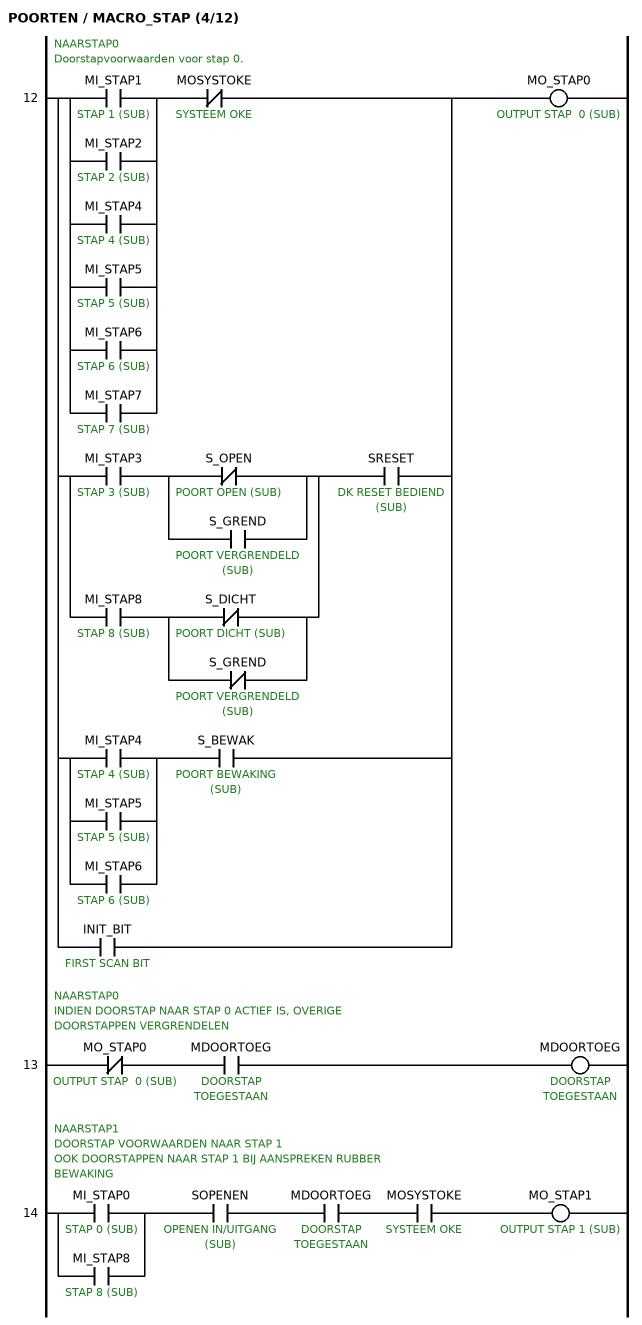
; [picture p469: POORTEN / MACRO_STAP, rungs 12-14]
; rung 12: NAARSTAP0 / Doorstapvoorwaarden voor stap 0.
LD MI_STAP1  ; STAP 1 (SUB)
OR MI_STAP2  ; STAP 2 (SUB)
OR MI_STAP4  ; STAP 4 (SUB)
OR MI_STAP5  ; STAP 5 (SUB)
OR MI_STAP6  ; STAP 6 (SUB)
OR MI_STAP7  ; STAP 7 (SUB)
ANDNOT MOSYSTOKE  ; SYSTEEM OKE
LD MI_STAP3  ; STAP 3 (SUB)
LDNOT S_OPEN  ; POORT OPEN (SUB)
OR S_GREND  ; POORT VERGRENDELD  (SUB)
ANDLD
LD MI_STAP8  ; STAP 8 (SUB)
LDNOT S_DICHT  ; POORT DICHT (SUB)
ORNOT S_GREND  ; POORT VERGRENDELD  (SUB)
ANDLD
ORLD
AND SRESET  ; DK RESET BEDIEND (SUB)
ORLD
LD MI_STAP4  ; STAP 4 (SUB)
OR MI_STAP5  ; STAP 5 (SUB)
OR MI_STAP6  ; STAP 6 (SUB)
AND S_BEWAK  ; POORT BEWAKING  (SUB)
ORLD
OR INIT_BIT  ; FIRST SCAN BIT
OUT MO_STAP0  ; OUTPUT STAP  0 (SUB)
; rung 13: NAARSTAP0 / INDIEN DOORSTAP NAAR STAP 0 ACTIEF IS, OVERIGE / DOORSTAPPEN VERGRENDELEN
LDNOT MO_STAP0  ; OUTPUT STAP  0 (SUB)
AND MDOORTOEG  ; DOORSTAP TOEGESTAAN
OUT MDOORTOEG  ; DOORSTAP TOEGESTAAN
; rung 14: NAARSTAP1 / DOORSTAP VOORWAARDEN NAAR STAP 1 / OOK DOORSTAPPEN NAAR STAP 1 BIJ AANSPREKEN RUBBER / BEWAKING
LD MI_STAP0  ; STAP 0 (SUB)
OR MI_STAP8  ; STAP 8 (SUB)
AND SOPENEN  ; OPENEN IN/UITGANG (SUB)
AND MDOORTOEG  ; DOORSTAP TOEGESTAAN
AND MOSYSTOKE  ; SYSTEEM OKE
OUT MO_STAP1  ; OUTPUT STAP 1 (SUB)

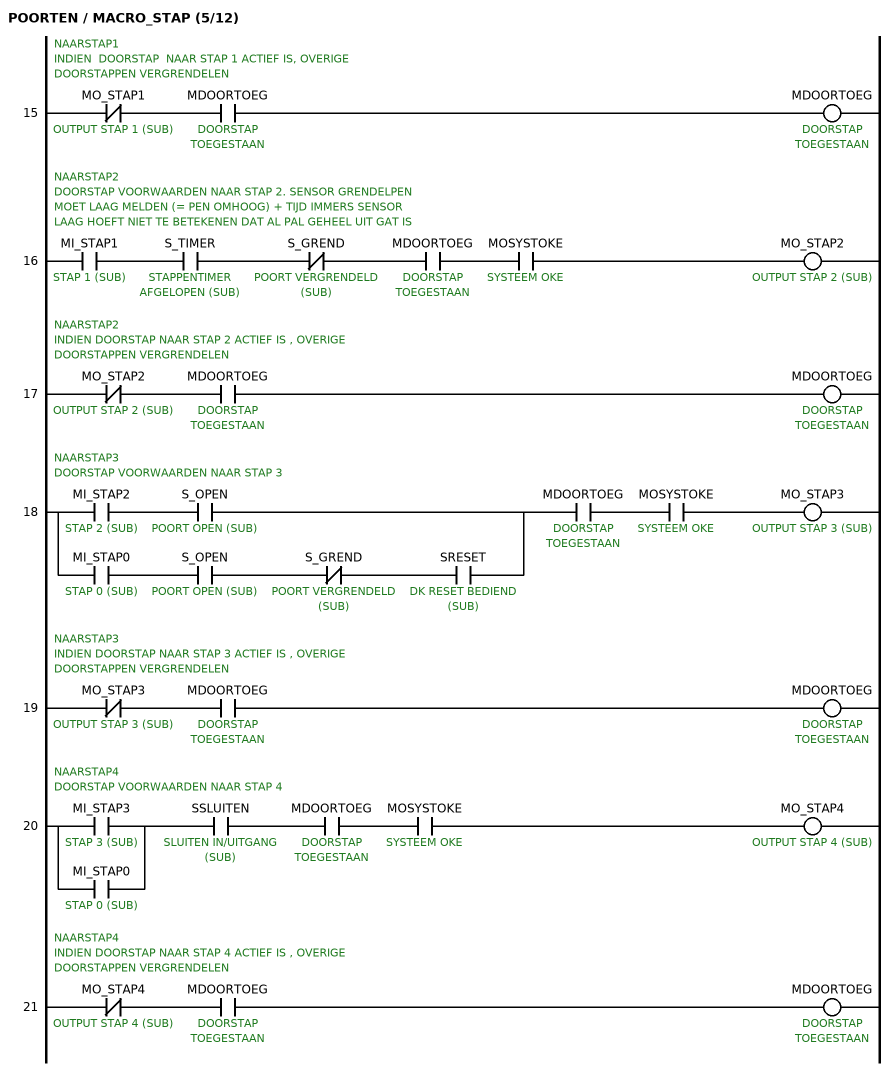
; rung 15: NAARSTAP1 / INDIEN  DOORSTAP  NAAR STAP 1 ACTIEF IS, OVERIGE / DOORSTAPPEN VERGRENDELEN
LDNOT MO_STAP1  ; OUTPUT STAP 1 (SUB)
AND MDOORTOEG  ; DOORSTAP TOEGESTAAN
OUT MDOORTOEG  ; DOORSTAP TOEGESTAAN
; rung 16: NAARSTAP2 / DOORSTAP VOORWAARDEN NAAR STAP 2. SENSOR GRENDELPEN / MOET LAAG MELDEN (= PEN OMHOOG) + TIJD IMMERS SENSOR / LAAG HOEFT NIET TE BETEKENEN DAT AL PAL GEHEEL UIT GAT IS
LD MI_STAP1  ; STAP 1 (SUB)
AND S_TIMER  ; STAPPENTIMER AFGELOPEN (SUB)
ANDNOT S_GREND  ; POORT VERGRENDELD  (SUB)
AND MDOORTOEG  ; DOORSTAP TOEGESTAAN
AND MOSYSTOKE  ; SYSTEEM OKE
OUT MO_STAP2  ; OUTPUT STAP 2 (SUB)
; rung 17: NAARSTAP2 / INDIEN DOORSTAP NAAR STAP 2 ACTIEF IS , OVERIGE / DOORSTAPPEN VERGRENDELEN
LDNOT MO_STAP2  ; OUTPUT STAP 2 (SUB)
AND MDOORTOEG  ; DOORSTAP TOEGESTAAN
OUT MDOORTOEG  ; DOORSTAP TOEGESTAAN
; rung 18: NAARSTAP3 / DOORSTAP VOORWAARDEN NAAR STAP 3
LD MI_STAP2  ; STAP 2 (SUB)
AND S_OPEN  ; POORT OPEN (SUB)
LD MI_STAP0  ; STAP 0 (SUB)
AND S_OPEN  ; POORT OPEN (SUB)
ANDNOT S_GREND  ; POORT VERGRENDELD  (SUB)
AND SRESET  ; DK RESET BEDIEND (SUB)
ORLD
AND MDOORTOEG  ; DOORSTAP TOEGESTAAN
AND MOSYSTOKE  ; SYSTEEM OKE
OUT MO_STAP3  ; OUTPUT STAP 3 (SUB)
; rung 19: NAARSTAP3 / INDIEN DOORSTAP NAAR STAP 3 ACTIEF IS , OVERIGE / DOORSTAPPEN VERGRENDELEN
LDNOT MO_STAP3  ; OUTPUT STAP 3 (SUB)
AND MDOORTOEG  ; DOORSTAP TOEGESTAAN
OUT MDOORTOEG  ; DOORSTAP TOEGESTAAN
; rung 20: NAARSTAP4 / DOORSTAP VOORWAARDEN NAAR STAP 4
LD MI_STAP3  ; STAP 3 (SUB)
OR MI_STAP0  ; STAP 0 (SUB)
AND SSLUITEN  ; SLUITEN IN/UITGANG (SUB)
AND MDOORTOEG  ; DOORSTAP TOEGESTAAN
AND MOSYSTOKE  ; SYSTEEM OKE
OUT MO_STAP4  ; OUTPUT STAP 4 (SUB)
; rung 21: NAARSTAP4 / INDIEN DOORSTAP NAAR STAP 4 ACTIEF IS , OVERIGE / DOORSTAPPEN VERGRENDELEN
LDNOT MO_STAP4  ; OUTPUT STAP 4 (SUB)
AND MDOORTOEG  ; DOORSTAP TOEGESTAAN
OUT MDOORTOEG  ; DOORSTAP TOEGESTAAN

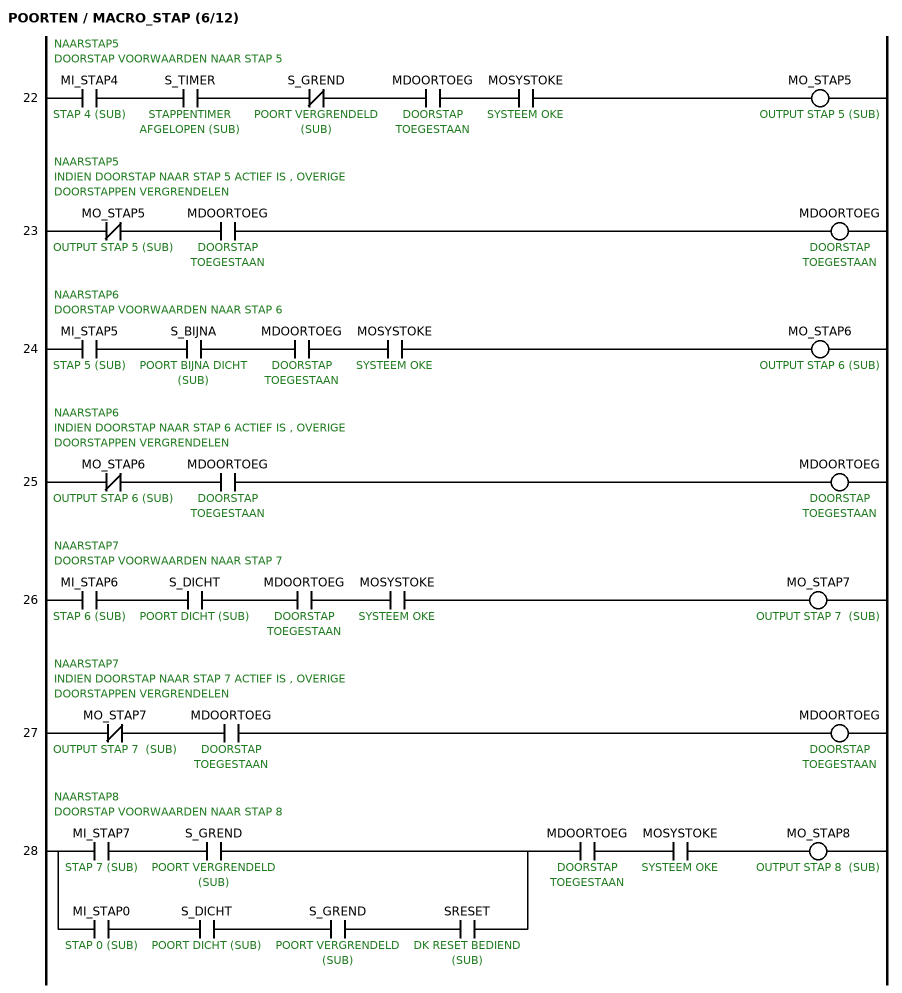
; rung 22: NAARSTAP5 / DOORSTAP VOORWAARDEN NAAR STAP 5
LD MI_STAP4  ; STAP 4 (SUB)
AND S_TIMER  ; STAPPENTIMER AFGELOPEN (SUB)
ANDNOT S_GREND  ; POORT VERGRENDELD  (SUB)
AND MDOORTOEG  ; DOORSTAP TOEGESTAAN
AND MOSYSTOKE  ; SYSTEEM OKE
OUT MO_STAP5  ; OUTPUT STAP 5 (SUB)
; rung 23: NAARSTAP5 / INDIEN DOORSTAP NAAR STAP 5 ACTIEF IS , OVERIGE / DOORSTAPPEN VERGRENDELEN
LDNOT MO_STAP5  ; OUTPUT STAP 5 (SUB)
AND MDOORTOEG  ; DOORSTAP TOEGESTAAN
OUT MDOORTOEG  ; DOORSTAP TOEGESTAAN
; rung 24: NAARSTAP6 / DOORSTAP VOORWAARDEN NAAR STAP 6
LD MI_STAP5  ; STAP 5 (SUB)
AND S_BIJNA  ; POORT BIJNA DICHT (SUB)
AND MDOORTOEG  ; DOORSTAP TOEGESTAAN
AND MOSYSTOKE  ; SYSTEEM OKE
OUT MO_STAP6  ; OUTPUT STAP 6 (SUB)
; rung 25: NAARSTAP6 / INDIEN DOORSTAP NAAR STAP 6 ACTIEF IS , OVERIGE / DOORSTAPPEN VERGRENDELEN
LDNOT MO_STAP6  ; OUTPUT STAP 6 (SUB)
AND MDOORTOEG  ; DOORSTAP TOEGESTAAN
OUT MDOORTOEG  ; DOORSTAP TOEGESTAAN
; rung 26: NAARSTAP7 / DOORSTAP VOORWAARDEN NAAR STAP 7
LD MI_STAP6  ; STAP 6 (SUB)
AND S_DICHT  ; POORT DICHT (SUB)
AND MDOORTOEG  ; DOORSTAP TOEGESTAAN
AND MOSYSTOKE  ; SYSTEEM OKE
OUT MO_STAP7  ; OUTPUT STAP 7  (SUB)
; rung 27: NAARSTAP7 / INDIEN DOORSTAP NAAR STAP 7 ACTIEF IS , OVERIGE / DOORSTAPPEN VERGRENDELEN
LDNOT MO_STAP7  ; OUTPUT STAP 7  (SUB)
AND MDOORTOEG  ; DOORSTAP TOEGESTAAN
OUT MDOORTOEG  ; DOORSTAP TOEGESTAAN
; rung 28: NAARSTAP8 / DOORSTAP VOORWAARDEN NAAR STAP 8
LD MI_STAP7  ; STAP 7 (SUB)
AND S_GREND  ; POORT VERGRENDELD  (SUB)
LD MI_STAP0  ; STAP 0 (SUB)
AND S_DICHT  ; POORT DICHT (SUB)
AND S_GREND  ; POORT VERGRENDELD  (SUB)
AND SRESET  ; DK RESET BEDIEND (SUB)
ORLD
AND MDOORTOEG  ; DOORSTAP TOEGESTAAN
AND MOSYSTOKE  ; SYSTEEM OKE
OUT MO_STAP8  ; OUTPUT STAP 8  (SUB)

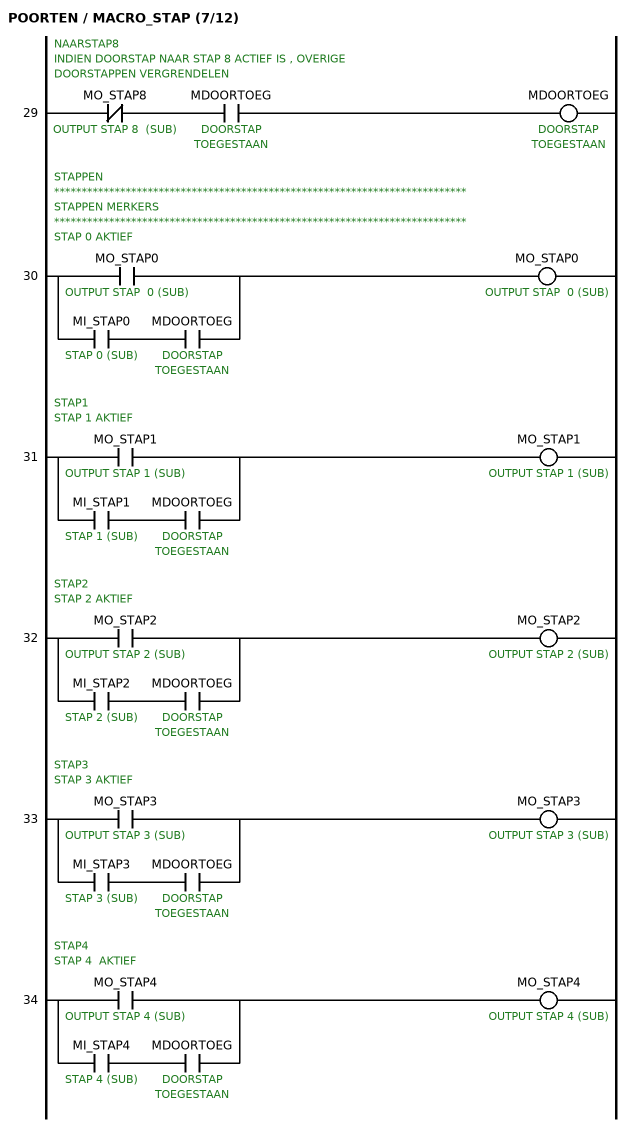
; rung 29: NAARSTAP8 / INDIEN DOORSTAP NAAR STAP 8 ACTIEF IS , OVERIGE / DOORSTAPPEN VERGRENDELEN
LDNOT MO_STAP8  ; OUTPUT STAP 8  (SUB)
AND MDOORTOEG  ; DOORSTAP TOEGESTAAN
OUT MDOORTOEG  ; DOORSTAP TOEGESTAAN
; rung 30: STAPPEN / *************************************************************************** / STAPPEN MERKERS / *************************************************************************** / STAP 0 AKTIEF
LD MO_STAP0  ; OUTPUT STAP  0 (SUB)
LD MI_STAP0  ; STAP 0 (SUB)
AND MDOORTOEG  ; DOORSTAP TOEGESTAAN
ORLD
OUT MO_STAP0  ; OUTPUT STAP  0 (SUB)
; rung 31: STAP1 / STAP 1 AKTIEF
LD MO_STAP1  ; OUTPUT STAP 1 (SUB)
LD MI_STAP1  ; STAP 1 (SUB)
AND MDOORTOEG  ; DOORSTAP TOEGESTAAN
ORLD
OUT MO_STAP1  ; OUTPUT STAP 1 (SUB)
; rung 32: STAP2 / STAP 2 AKTIEF
LD MO_STAP2  ; OUTPUT STAP 2 (SUB)
LD MI_STAP2  ; STAP 2 (SUB)
AND MDOORTOEG  ; DOORSTAP TOEGESTAAN
ORLD
OUT MO_STAP2  ; OUTPUT STAP 2 (SUB)
; rung 33: STAP3 / STAP 3 AKTIEF
LD MO_STAP3  ; OUTPUT STAP 3 (SUB)
LD MI_STAP3  ; STAP 3 (SUB)
AND MDOORTOEG  ; DOORSTAP TOEGESTAAN
ORLD
OUT MO_STAP3  ; OUTPUT STAP 3 (SUB)
; rung 34: STAP4 / STAP 4  AKTIEF
LD MO_STAP4  ; OUTPUT STAP 4 (SUB)
LD MI_STAP4  ; STAP 4 (SUB)
AND MDOORTOEG  ; DOORSTAP TOEGESTAAN
ORLD
OUT MO_STAP4  ; OUTPUT STAP 4 (SUB)

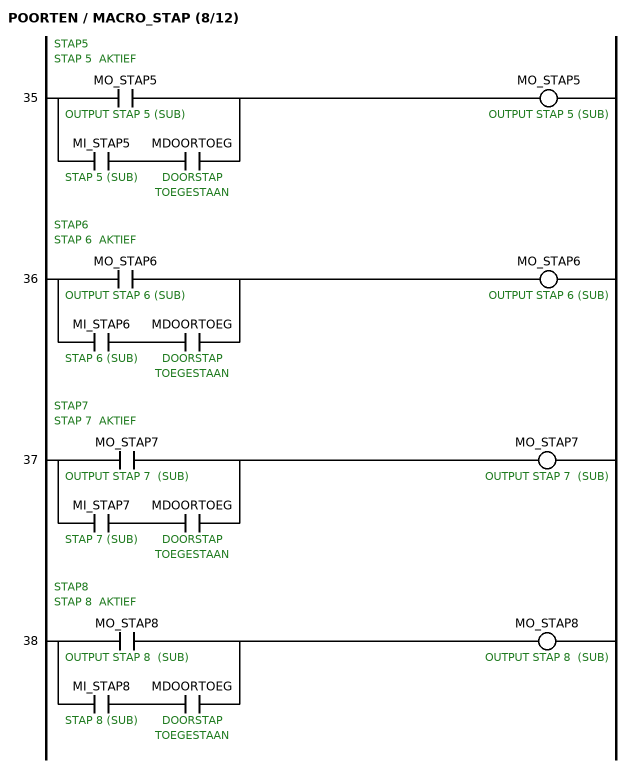
; rung 35: STAP5 / STAP 5  AKTIEF
LD MO_STAP5  ; OUTPUT STAP 5 (SUB)
LD MI_STAP5  ; STAP 5 (SUB)
AND MDOORTOEG  ; DOORSTAP TOEGESTAAN
ORLD
OUT MO_STAP5  ; OUTPUT STAP 5 (SUB)
; rung 36: STAP6 / STAP 6  AKTIEF
LD MO_STAP6  ; OUTPUT STAP 6 (SUB)
LD MI_STAP6  ; STAP 6 (SUB)
AND MDOORTOEG  ; DOORSTAP TOEGESTAAN
ORLD
OUT MO_STAP6  ; OUTPUT STAP 6 (SUB)
; rung 37: STAP7 / STAP 7  AKTIEF
LD MO_STAP7  ; OUTPUT STAP 7  (SUB)
LD MI_STAP7  ; STAP 7 (SUB)
AND MDOORTOEG  ; DOORSTAP TOEGESTAAN
ORLD
OUT MO_STAP7  ; OUTPUT STAP 7  (SUB)
; rung 38: STAP8 / STAP 8  AKTIEF
LD MO_STAP8  ; OUTPUT STAP 8  (SUB)
LD MI_STAP8  ; STAP 8 (SUB)
AND MDOORTOEG  ; DOORSTAP TOEGESTAAN
ORLD
OUT MO_STAP8  ; OUTPUT STAP 8  (SUB)

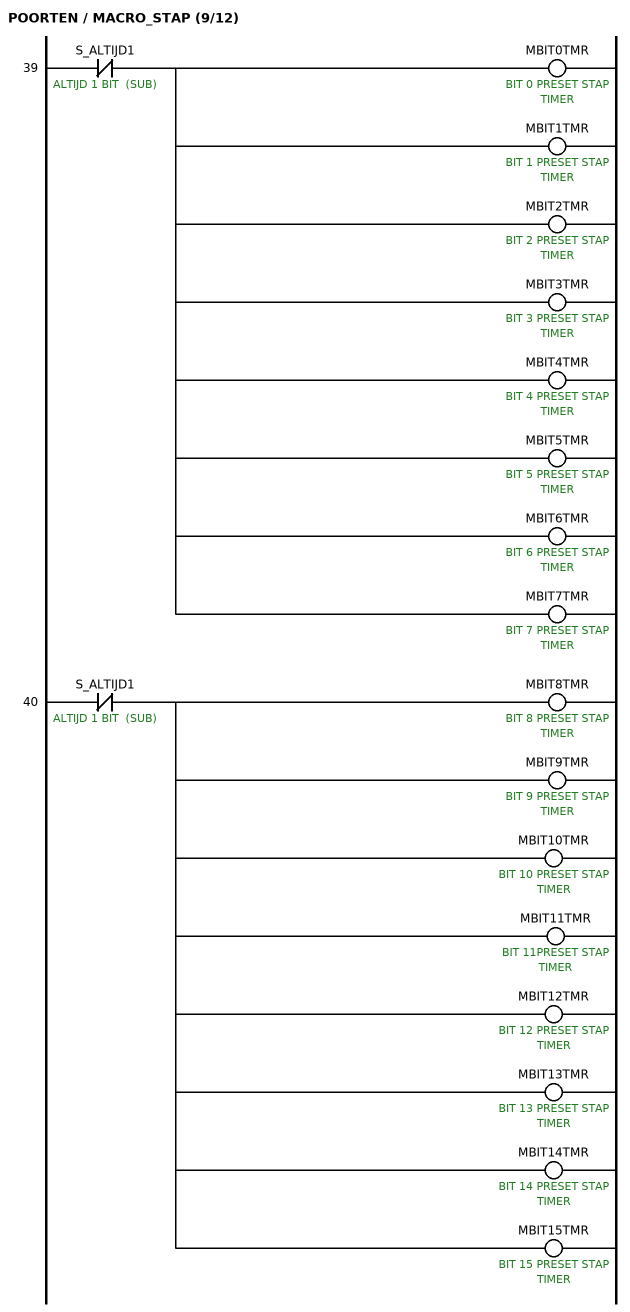
; rung 39
LDNOT S_ALTIJD1  ; ALTIJD 1 BIT  (SUB)
OUT MBIT0TMR  ; BIT 0 PRESET STAP TIMER
OUT MBIT1TMR  ; BIT 1 PRESET STAP TIMER
OUT MBIT2TMR  ; BIT 2 PRESET STAP TIMER
OUT MBIT3TMR  ; BIT 3 PRESET STAP TIMER
OUT MBIT4TMR  ; BIT 4 PRESET STAP TIMER
OUT MBIT5TMR  ; BIT 5 PRESET STAP TIMER
OUT MBIT6TMR  ; BIT 6 PRESET STAP TIMER
OUT MBIT7TMR  ; BIT 7 PRESET STAP TIMER
; rung 40
LDNOT S_ALTIJD1  ; ALTIJD 1 BIT  (SUB)
OUT MBIT8TMR  ; BIT 8 PRESET STAP TIMER
OUT MBIT9TMR  ; BIT 9 PRESET STAP TIMER
OUT MBIT10TMR  ; BIT 10 PRESET STAP TIMER
OUT MBIT11TMR  ; BIT 11PRESET STAP TIMER
OUT MBIT12TMR  ; BIT 12 PRESET STAP TIMER
OUT MBIT13TMR  ; BIT 13 PRESET STAP TIMER
OUT MBIT14TMR  ; BIT 14 PRESET STAP TIMER
OUT MBIT15TMR  ; BIT 15 PRESET STAP TIMER

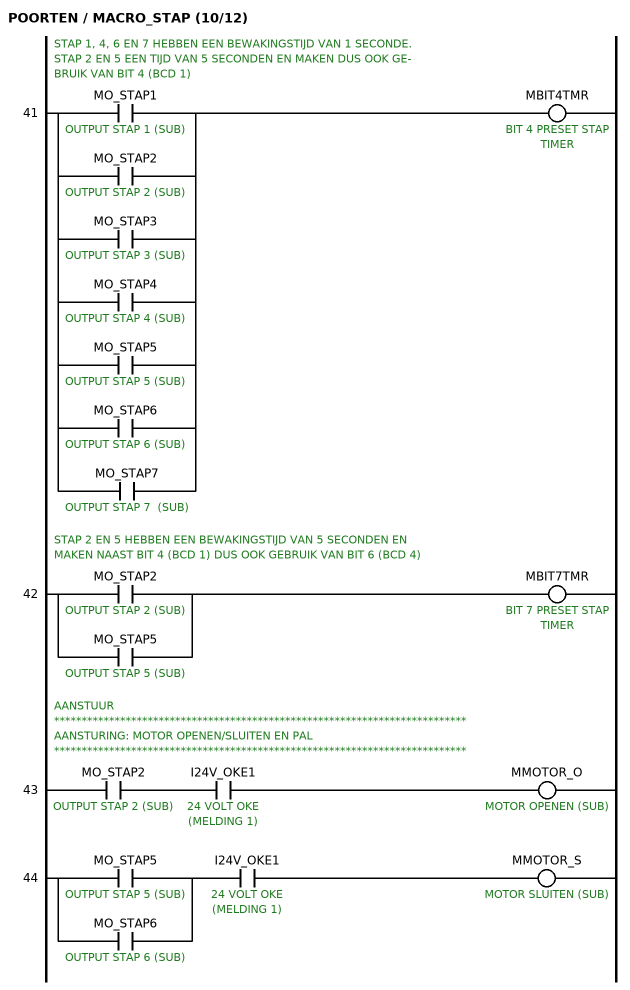
; rung 41: STAP 1, 4, 6 EN 7 HEBBEN EEN BEWAKINGSTIJD VAN 1 SECONDE. / STAP 2 EN 5 EEN TIJD VAN 5 SECONDEN EN MAKEN DUS OOK GE- / BRUIK VAN BIT 4 (BCD 1)
LD MO_STAP1  ; OUTPUT STAP 1 (SUB)
OR MO_STAP2  ; OUTPUT STAP 2 (SUB)
OR MO_STAP3  ; OUTPUT STAP 3 (SUB)
OR MO_STAP4  ; OUTPUT STAP 4 (SUB)
OR MO_STAP5  ; OUTPUT STAP 5 (SUB)
OR MO_STAP6  ; OUTPUT STAP 6 (SUB)
OR MO_STAP7  ; OUTPUT STAP 7  (SUB)
OUT MBIT4TMR  ; BIT 4 PRESET STAP TIMER
; rung 42: STAP 2 EN 5 HEBBEN EEN BEWAKINGSTIJD VAN 5 SECONDEN EN / MAKEN NAAST BIT 4 (BCD 1) DUS OOK GEBRUIK VAN BIT 6 (BCD 4)
LD MO_STAP2  ; OUTPUT STAP 2 (SUB)
OR MO_STAP5  ; OUTPUT STAP 5 (SUB)
OUT MBIT7TMR  ; BIT 7 PRESET STAP TIMER
; rung 43: AANSTUUR / *************************************************************************** / AANSTURING: MOTOR OPENEN/SLUITEN EN PAL / ***************************************************************************
LD MO_STAP2  ; OUTPUT STAP 2 (SUB)
AND I24V_OKE1  ; 24 VOLT OKE (MELDING 1)
OUT MMOTOR_O  ; MOTOR OPENEN (SUB)
; rung 44
LD MO_STAP5  ; OUTPUT STAP 5 (SUB)
OR MO_STAP6  ; OUTPUT STAP 6 (SUB)
AND I24V_OKE1  ; 24 VOLT OKE (MELDING 1)
OUT MMOTOR_S  ; MOTOR SLUITEN (SUB)

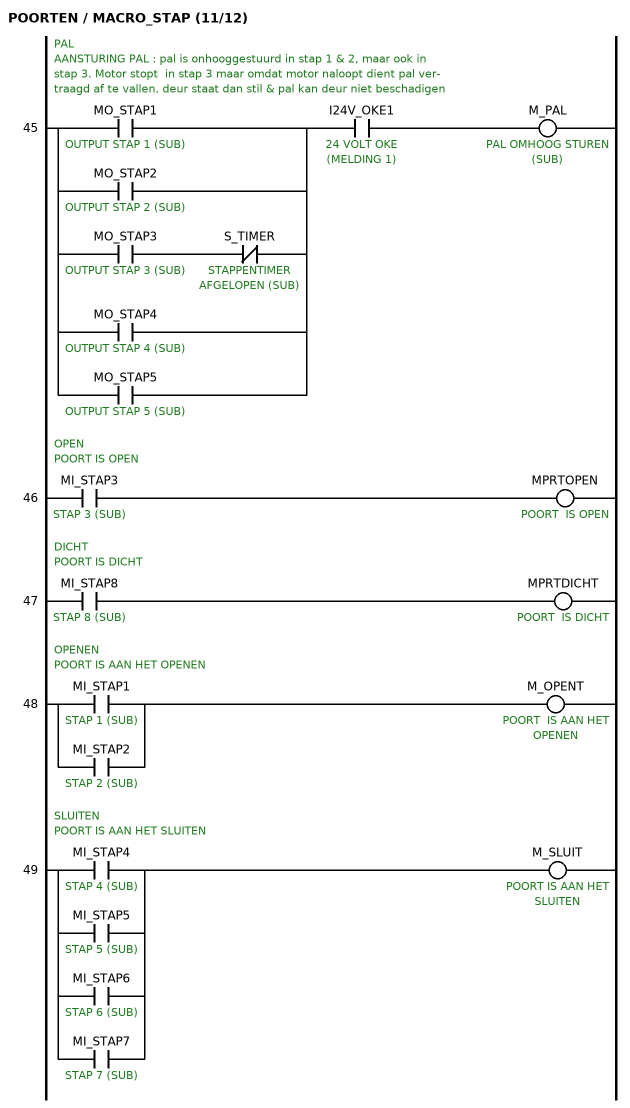
; rung 45: PAL / AANSTURING PAL : pal is onhooggestuurd in stap 1 & 2, maar ook in / stap 3. Motor stopt  in stap 3 maar omdat motor naloopt dient pal ver- / traagd af te vallen. deur staat dan stil & pal kan deur niet beschadigen
LD MO_STAP1  ; OUTPUT STAP 1 (SUB)
OR MO_STAP2  ; OUTPUT STAP 2 (SUB)
LD MO_STAP3  ; OUTPUT STAP 3 (SUB)
ANDNOT S_TIMER  ; STAPPENTIMER AFGELOPEN (SUB)
ORLD
OR MO_STAP4  ; OUTPUT STAP 4 (SUB)
OR MO_STAP5  ; OUTPUT STAP 5 (SUB)
AND I24V_OKE1  ; 24 VOLT OKE (MELDING 1)
OUT M_PAL  ; PAL OMHOOG STUREN (SUB)
; rung 46: OPEN / POORT IS OPEN
LD MI_STAP3  ; STAP 3 (SUB)
OUT MPRTOPEN  ; POORT  IS OPEN
; rung 47: DICHT / POORT IS DICHT
LD MI_STAP8  ; STAP 8 (SUB)
OUT MPRTDICHT  ; POORT  IS DICHT
; rung 48: OPENEN / POORT IS AAN HET OPENEN
LD MI_STAP1  ; STAP 1 (SUB)
OR MI_STAP2  ; STAP 2 (SUB)
OUT M_OPENT  ; POORT  IS AAN HET OPENEN
; rung 49: SLUITEN / POORT IS AAN HET SLUITEN
LD MI_STAP4  ; STAP 4 (SUB)
OR MI_STAP5  ; STAP 5 (SUB)
OR MI_STAP6  ; STAP 6 (SUB)
OR MI_STAP7  ; STAP 7 (SUB)
OUT M_SLUIT  ; POORT IS AAN HET SLUITEN

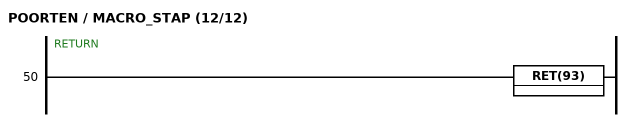
; rung 50: RETURN
RET(93)

### Section SUB_DISPLAY

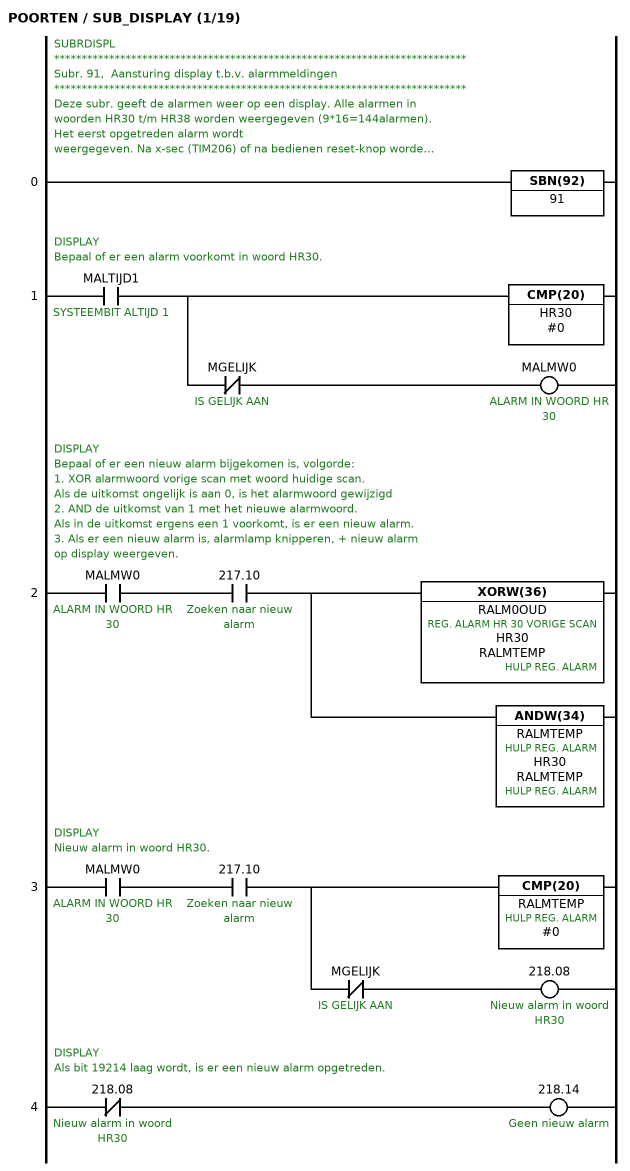
; rung 0: SUBRDISPL / *************************************************************************** / Subr. 91,  Aansturing display t.b.v. alarmmeldingen / *************************************************************************** / Deze subr. geeft de alarmen weer op een display. Alle alarmen in / woorden HR30 t/m HR38 worden weergegeven (9*16=144alarmen). / Het eerst opgetreden alarm wordt / weergegeven. Na x-sec (TIM206) of na bedienen reset-knop worden / alle alarmen gescrolld, met schroltijd TIM207. Als tijdens scrollen een / nieuw alarm optreedt, wordt dit alarm weer continu weergegeven.
SBN(92) 91
; rung 1: DISPLAY / Bepaal of er een alarm voorkomt in woord HR30.
LD MALTIJD1  ; SYSTEEMBIT ALTIJD 1
CMP(20) HR30 #0
ANDNOT MGELIJK  ; IS GELIJK AAN
OUT MALMW0  ; ALARM IN WOORD HR 30
; rung 2: DISPLAY / Bepaal of er een nieuw alarm bijgekomen is, volgorde: / 1. XOR alarmwoord vorige scan met woord huidige scan. / Als de uitkomst ongelijk is aan 0, is het alarmwoord gewijzigd / 2. AND de uitkomst van 1 met het nieuwe alarmwoord. / Als in de uitkomst ergens een 1 voorkomt, is er een nieuw alarm. / 3. Als er een nieuw alarm is, alarmlamp knipperen, + nieuw alarm / op display weergeven.
LD MALMW0  ; ALARM IN WOORD HR 30
AND 217.10  ; Zoeken naar nieuw alarm
XORW(36) RALM0OUD HR30 RALMTEMP  ; REG. ALARM HR 30 VORIGE SCAN, HULP REG. ALARM
ANDW(34) RALMTEMP HR30 RALMTEMP  ; HULP REG. ALARM
; rung 3: DISPLAY / Nieuw alarm in woord HR30.
LD MALMW0  ; ALARM IN WOORD HR 30
AND 217.10  ; Zoeken naar nieuw alarm
CMP(20) RALMTEMP #0  ; HULP REG. ALARM
ANDNOT MGELIJK  ; IS GELIJK AAN
OUT 218.08  ; Nieuw alarm in woord HR30
; rung 4: DISPLAY / Als bit 19214 laag wordt, is er een nieuw alarm opgetreden.
LDNOT 218.08  ; Nieuw alarm in woord HR30
OUT 218.14  ; Geen nieuw alarm

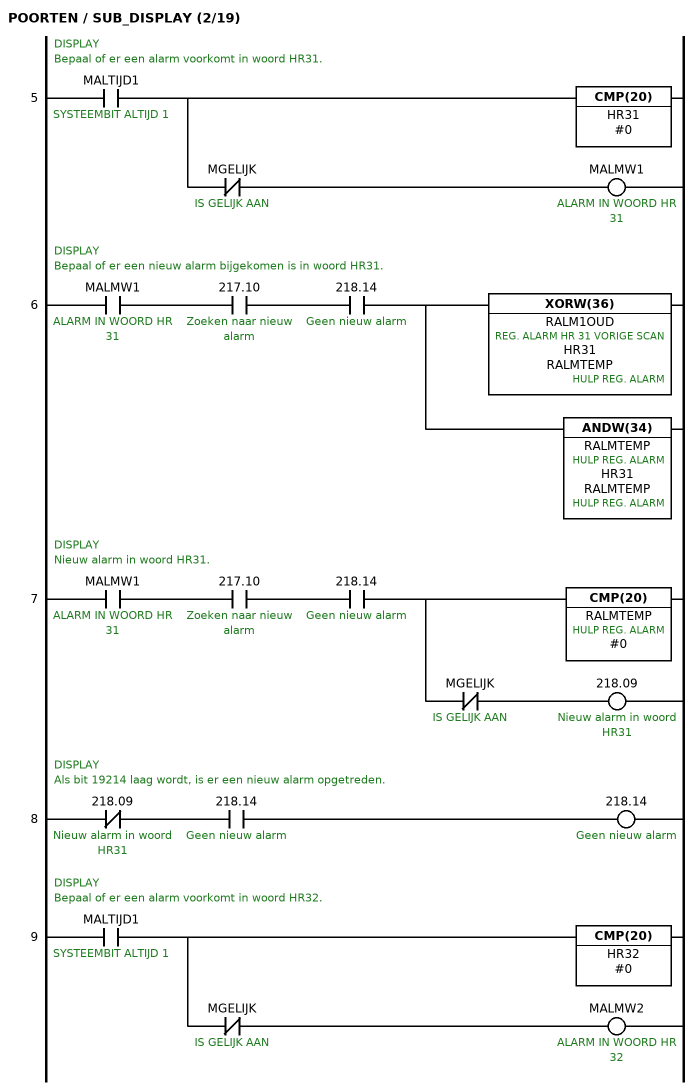
; rung 5: DISPLAY / Bepaal of er een alarm voorkomt in woord HR31.
LD MALTIJD1  ; SYSTEEMBIT ALTIJD 1
CMP(20) HR31 #0
ANDNOT MGELIJK  ; IS GELIJK AAN
OUT MALMW1  ; ALARM IN WOORD HR 31
; rung 6: DISPLAY / Bepaal of er een nieuw alarm bijgekomen is in woord HR31.
LD MALMW1  ; ALARM IN WOORD HR 31
AND 217.10  ; Zoeken naar nieuw alarm
AND 218.14  ; Geen nieuw alarm
XORW(36) RALM1OUD HR31 RALMTEMP  ; REG. ALARM HR 31 VORIGE SCAN, HULP REG. ALARM
ANDW(34) RALMTEMP HR31 RALMTEMP  ; HULP REG. ALARM
; rung 7: DISPLAY / Nieuw alarm in woord HR31.
LD MALMW1  ; ALARM IN WOORD HR 31
AND 217.10  ; Zoeken naar nieuw alarm
AND 218.14  ; Geen nieuw alarm
CMP(20) RALMTEMP #0  ; HULP REG. ALARM
ANDNOT MGELIJK  ; IS GELIJK AAN
OUT 218.09  ; Nieuw alarm in woord HR31
; rung 8: DISPLAY / Als bit 19214 laag wordt, is er een nieuw alarm opgetreden.
LDNOT 218.09  ; Nieuw alarm in woord HR31
AND 218.14  ; Geen nieuw alarm
OUT 218.14  ; Geen nieuw alarm
; rung 9: DISPLAY / Bepaal of er een alarm voorkomt in woord HR32.
LD MALTIJD1  ; SYSTEEMBIT ALTIJD 1
CMP(20) HR32 #0
ANDNOT MGELIJK  ; IS GELIJK AAN
OUT MALMW2  ; ALARM IN WOORD HR 32

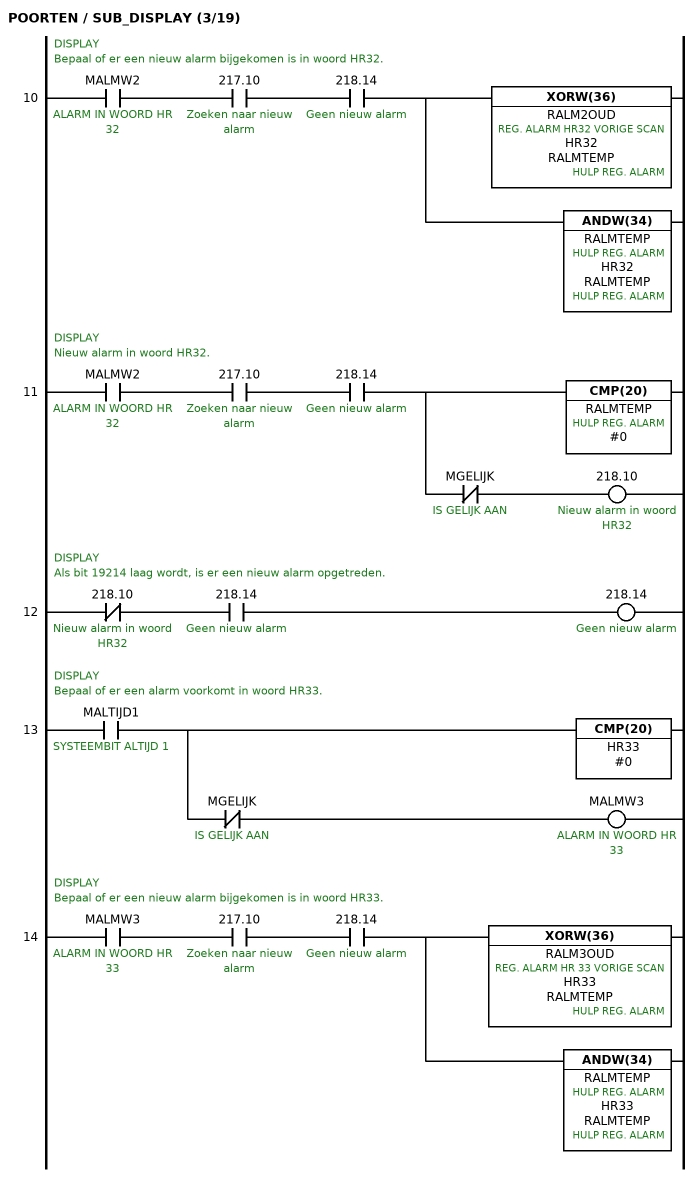
; rung 10: DISPLAY / Bepaal of er een nieuw alarm bijgekomen is in woord HR32.
LD MALMW2  ; ALARM IN WOORD HR 32
AND 217.10  ; Zoeken naar nieuw alarm
AND 218.14  ; Geen nieuw alarm
XORW(36) RALM2OUD HR32 RALMTEMP  ; REG. ALARM HR32 VORIGE SCAN, HULP REG. ALARM
ANDW(34) RALMTEMP HR32 RALMTEMP  ; HULP REG. ALARM
; rung 11: DISPLAY / Nieuw alarm in woord HR32.
LD MALMW2  ; ALARM IN WOORD HR 32
AND 217.10  ; Zoeken naar nieuw alarm
AND 218.14  ; Geen nieuw alarm
CMP(20) RALMTEMP #0  ; HULP REG. ALARM
ANDNOT MGELIJK  ; IS GELIJK AAN
OUT 218.10  ; Nieuw alarm in woord HR32
; rung 12: DISPLAY / Als bit 19214 laag wordt, is er een nieuw alarm opgetreden.
LDNOT 218.10  ; Nieuw alarm in woord HR32
AND 218.14  ; Geen nieuw alarm
OUT 218.14  ; Geen nieuw alarm
; rung 13: DISPLAY / Bepaal of er een alarm voorkomt in woord HR33.
LD MALTIJD1  ; SYSTEEMBIT ALTIJD 1
CMP(20) HR33 #0
ANDNOT MGELIJK  ; IS GELIJK AAN
OUT MALMW3  ; ALARM IN WOORD HR 33
; rung 14: DISPLAY / Bepaal of er een nieuw alarm bijgekomen is in woord HR33.
LD MALMW3  ; ALARM IN WOORD HR 33
AND 217.10  ; Zoeken naar nieuw alarm
AND 218.14  ; Geen nieuw alarm
XORW(36) RALM3OUD HR33 RALMTEMP  ; REG. ALARM HR 33 VORIGE SCAN, HULP REG. ALARM
ANDW(34) RALMTEMP HR33 RALMTEMP  ; HULP REG. ALARM

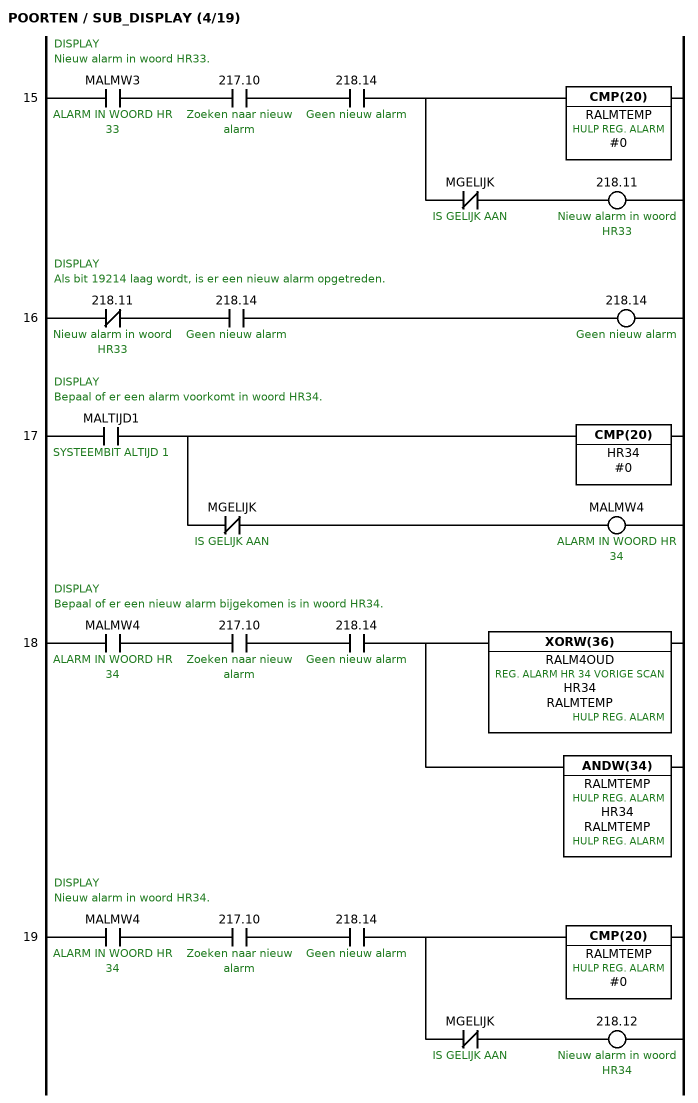
; rung 15: DISPLAY / Nieuw alarm in woord HR33.
LD MALMW3  ; ALARM IN WOORD HR 33
AND 217.10  ; Zoeken naar nieuw alarm
AND 218.14  ; Geen nieuw alarm
CMP(20) RALMTEMP #0  ; HULP REG. ALARM
ANDNOT MGELIJK  ; IS GELIJK AAN
OUT 218.11  ; Nieuw alarm in woord HR33
; rung 16: DISPLAY / Als bit 19214 laag wordt, is er een nieuw alarm opgetreden.
LDNOT 218.11  ; Nieuw alarm in woord HR33
AND 218.14  ; Geen nieuw alarm
OUT 218.14  ; Geen nieuw alarm
; rung 17: DISPLAY / Bepaal of er een alarm voorkomt in woord HR34.
LD MALTIJD1  ; SYSTEEMBIT ALTIJD 1
CMP(20) HR34 #0
ANDNOT MGELIJK  ; IS GELIJK AAN
OUT MALMW4  ; ALARM IN WOORD HR 34
; rung 18: DISPLAY / Bepaal of er een nieuw alarm bijgekomen is in woord HR34.
LD MALMW4  ; ALARM IN WOORD HR 34
AND 217.10  ; Zoeken naar nieuw alarm
AND 218.14  ; Geen nieuw alarm
XORW(36) RALM4OUD HR34 RALMTEMP  ; REG. ALARM HR 34 VORIGE SCAN, HULP REG. ALARM
ANDW(34) RALMTEMP HR34 RALMTEMP  ; HULP REG. ALARM
; rung 19: DISPLAY / Nieuw alarm in woord HR34.
LD MALMW4  ; ALARM IN WOORD HR 34
AND 217.10  ; Zoeken naar nieuw alarm
AND 218.14  ; Geen nieuw alarm
CMP(20) RALMTEMP #0  ; HULP REG. ALARM
ANDNOT MGELIJK  ; IS GELIJK AAN
OUT 218.12  ; Nieuw alarm in woord HR34

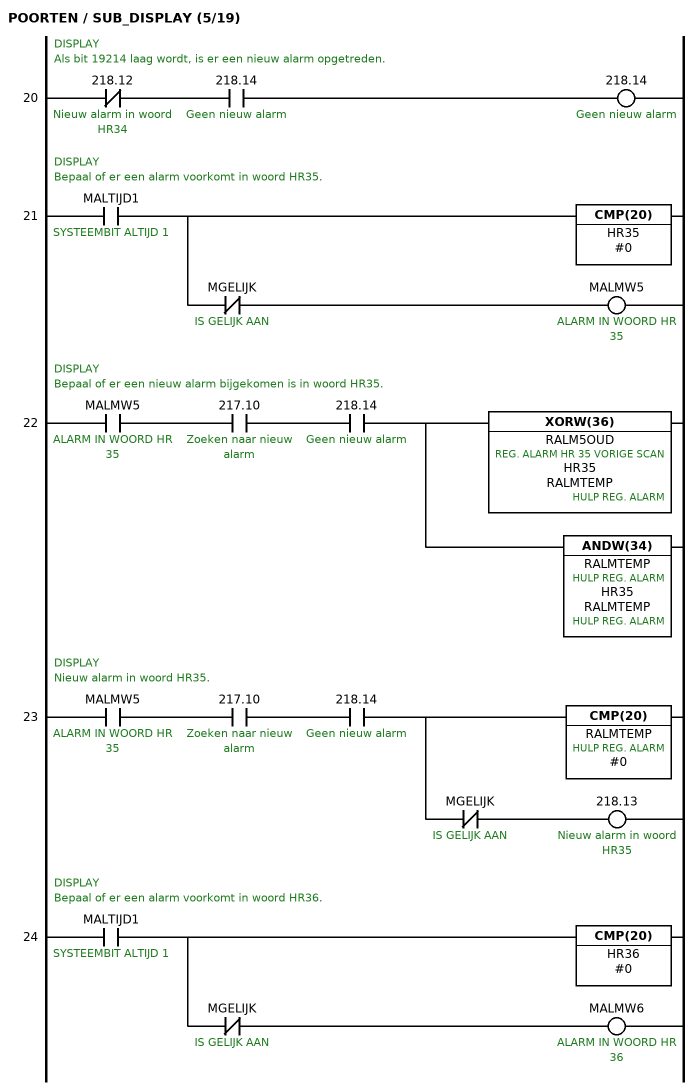
; rung 20: DISPLAY / Als bit 19214 laag wordt, is er een nieuw alarm opgetreden.
LDNOT 218.12  ; Nieuw alarm in woord HR34
AND 218.14  ; Geen nieuw alarm
OUT 218.14  ; Geen nieuw alarm
; rung 21: DISPLAY / Bepaal of er een alarm voorkomt in woord HR35.
LD MALTIJD1  ; SYSTEEMBIT ALTIJD 1
CMP(20) HR35 #0
ANDNOT MGELIJK  ; IS GELIJK AAN
OUT MALMW5  ; ALARM IN WOORD HR 35
; rung 22: DISPLAY / Bepaal of er een nieuw alarm bijgekomen is in woord HR35.
LD MALMW5  ; ALARM IN WOORD HR 35
AND 217.10  ; Zoeken naar nieuw alarm
AND 218.14  ; Geen nieuw alarm
XORW(36) RALM5OUD HR35 RALMTEMP  ; REG. ALARM HR 35 VORIGE SCAN, HULP REG. ALARM
ANDW(34) RALMTEMP HR35 RALMTEMP  ; HULP REG. ALARM
; rung 23: DISPLAY / Nieuw alarm in woord HR35.
LD MALMW5  ; ALARM IN WOORD HR 35
AND 217.10  ; Zoeken naar nieuw alarm
AND 218.14  ; Geen nieuw alarm
CMP(20) RALMTEMP #0  ; HULP REG. ALARM
ANDNOT MGELIJK  ; IS GELIJK AAN
OUT 218.13  ; Nieuw alarm in woord HR35
; rung 24: DISPLAY / Bepaal of er een alarm voorkomt in woord HR36.
LD MALTIJD1  ; SYSTEEMBIT ALTIJD 1
CMP(20) HR36 #0
ANDNOT MGELIJK  ; IS GELIJK AAN
OUT MALMW6  ; ALARM IN WOORD HR 36

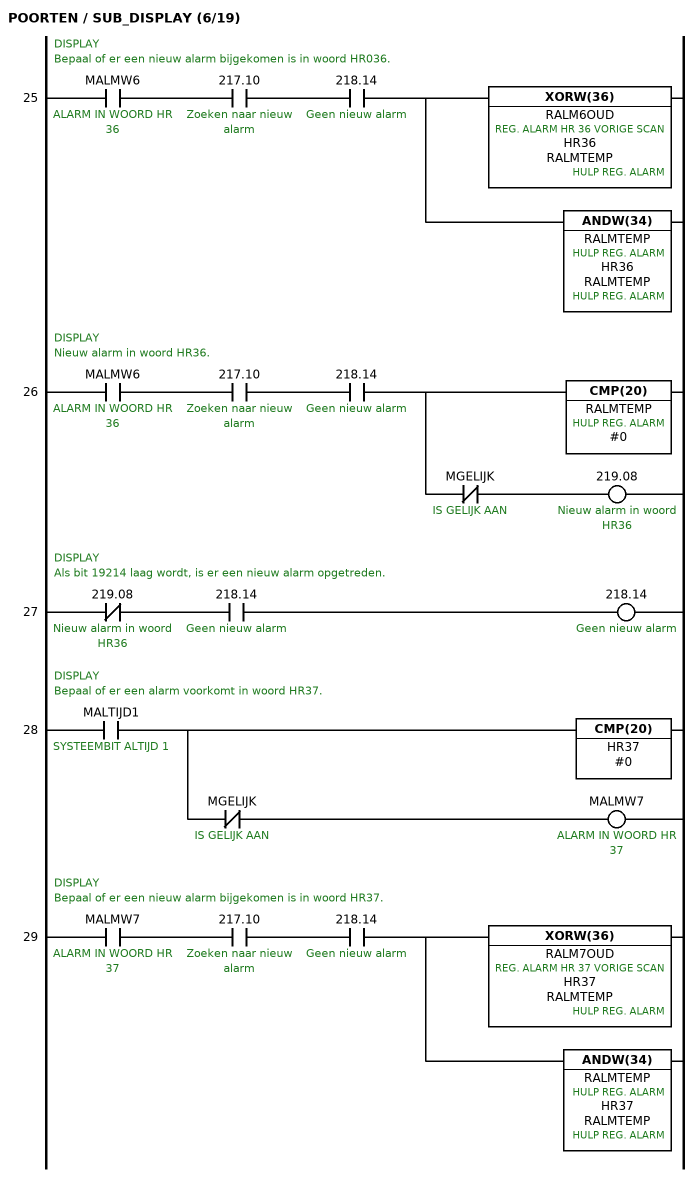
; rung 25: DISPLAY / Bepaal of er een nieuw alarm bijgekomen is in woord HR036.
LD MALMW6  ; ALARM IN WOORD HR 36
AND 217.10  ; Zoeken naar nieuw alarm
AND 218.14  ; Geen nieuw alarm
XORW(36) RALM6OUD HR36 RALMTEMP  ; REG. ALARM HR 36 VORIGE SCAN, HULP REG. ALARM
ANDW(34) RALMTEMP HR36 RALMTEMP  ; HULP REG. ALARM
; rung 26: DISPLAY / Nieuw alarm in woord HR36.
LD MALMW6  ; ALARM IN WOORD HR 36
AND 217.10  ; Zoeken naar nieuw alarm
AND 218.14  ; Geen nieuw alarm
CMP(20) RALMTEMP #0  ; HULP REG. ALARM
ANDNOT MGELIJK  ; IS GELIJK AAN
OUT 219.08  ; Nieuw alarm in woord HR36
; rung 27: DISPLAY / Als bit 19214 laag wordt, is er een nieuw alarm opgetreden.
LDNOT 219.08  ; Nieuw alarm in woord HR36
AND 218.14  ; Geen nieuw alarm
OUT 218.14  ; Geen nieuw alarm
; rung 28: DISPLAY / Bepaal of er een alarm voorkomt in woord HR37.
LD MALTIJD1  ; SYSTEEMBIT ALTIJD 1
CMP(20) HR37 #0
ANDNOT MGELIJK  ; IS GELIJK AAN
OUT MALMW7  ; ALARM IN WOORD HR 37
; rung 29: DISPLAY / Bepaal of er een nieuw alarm bijgekomen is in woord HR37.
LD MALMW7  ; ALARM IN WOORD HR 37
AND 217.10  ; Zoeken naar nieuw alarm
AND 218.14  ; Geen nieuw alarm
XORW(36) RALM7OUD HR37 RALMTEMP  ; REG. ALARM HR 37 VORIGE SCAN, HULP REG. ALARM
ANDW(34) RALMTEMP HR37 RALMTEMP  ; HULP REG. ALARM

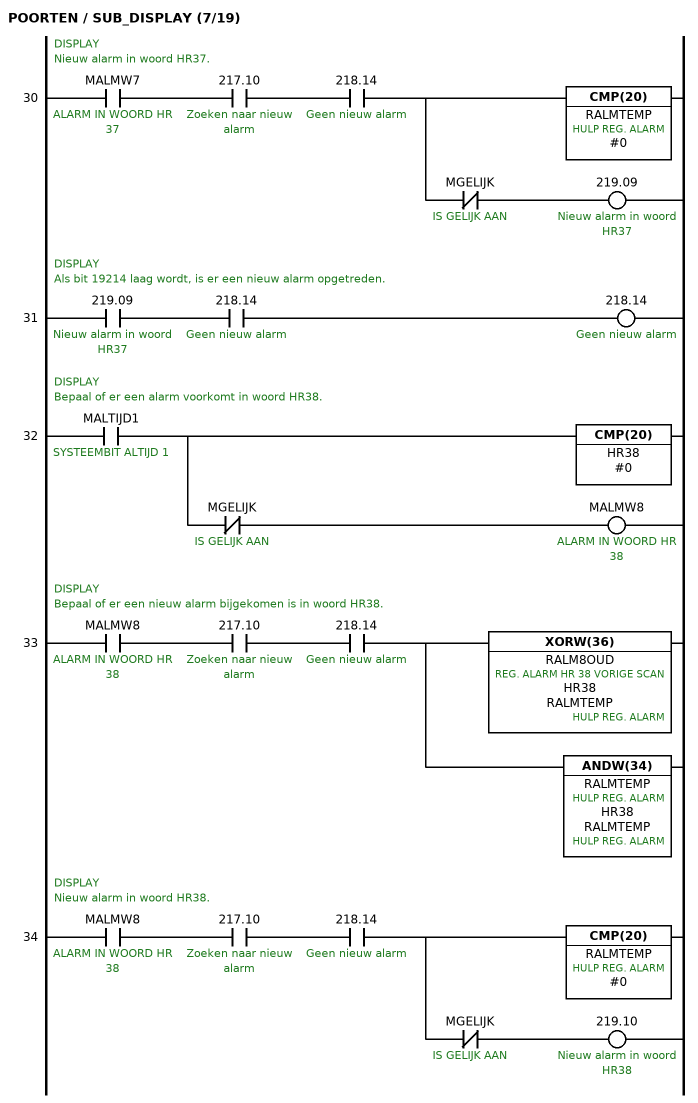
; rung 30: DISPLAY / Nieuw alarm in woord HR37.
LD MALMW7  ; ALARM IN WOORD HR 37
AND 217.10  ; Zoeken naar nieuw alarm
AND 218.14  ; Geen nieuw alarm
CMP(20) RALMTEMP #0  ; HULP REG. ALARM
ANDNOT MGELIJK  ; IS GELIJK AAN
OUT 219.09  ; Nieuw alarm in woord HR37
; rung 31: DISPLAY / Als bit 19214 laag wordt, is er een nieuw alarm opgetreden.
LD 219.09  ; Nieuw alarm in woord HR37
AND 218.14  ; Geen nieuw alarm
OUT 218.14  ; Geen nieuw alarm
; rung 32: DISPLAY / Bepaal of er een alarm voorkomt in woord HR38.
LD MALTIJD1  ; SYSTEEMBIT ALTIJD 1
CMP(20) HR38 #0
ANDNOT MGELIJK  ; IS GELIJK AAN
OUT MALMW8  ; ALARM IN WOORD HR 38
; rung 33: DISPLAY / Bepaal of er een nieuw alarm bijgekomen is in woord HR38.
LD MALMW8  ; ALARM IN WOORD HR 38
AND 217.10  ; Zoeken naar nieuw alarm
AND 218.14  ; Geen nieuw alarm
XORW(36) RALM8OUD HR38 RALMTEMP  ; REG. ALARM HR 38 VORIGE SCAN, HULP REG. ALARM
ANDW(34) RALMTEMP HR38 RALMTEMP  ; HULP REG. ALARM
; rung 34: DISPLAY / Nieuw alarm in woord HR38.
LD MALMW8  ; ALARM IN WOORD HR 38
AND 217.10  ; Zoeken naar nieuw alarm
AND 218.14  ; Geen nieuw alarm
CMP(20) RALMTEMP #0  ; HULP REG. ALARM
ANDNOT MGELIJK  ; IS GELIJK AAN
OUT 219.10  ; Nieuw alarm in woord HR38

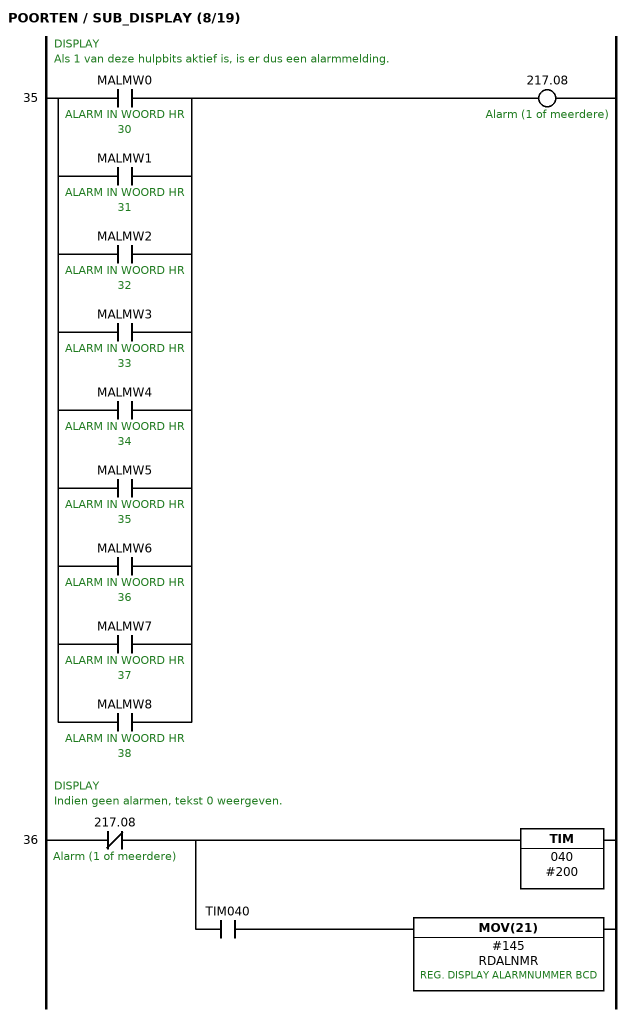
; rung 35: DISPLAY / Als 1 van deze hulpbits aktief is, is er dus een alarmmelding.
LD MALMW0  ; ALARM IN WOORD HR 30
OR MALMW1  ; ALARM IN WOORD HR 31
OR MALMW2  ; ALARM IN WOORD HR 32
OR MALMW3  ; ALARM IN WOORD HR 33
OR MALMW4  ; ALARM IN WOORD HR 34
OR MALMW5  ; ALARM IN WOORD HR 35
OR MALMW6  ; ALARM IN WOORD HR 36
OR MALMW7  ; ALARM IN WOORD HR 37
OR MALMW8  ; ALARM IN WOORD HR 38
OUT 217.08  ; Alarm (1 of meerdere)
; rung 36: DISPLAY / Indien geen alarmen, tekst 0 weergeven.
LDNOT 217.08  ; Alarm (1 of meerdere)
TIM 040 #200
AND TIM040
MOV(21) #145 RDALNMR  ; REG. DISPLAY ALARMNUMMER BCD

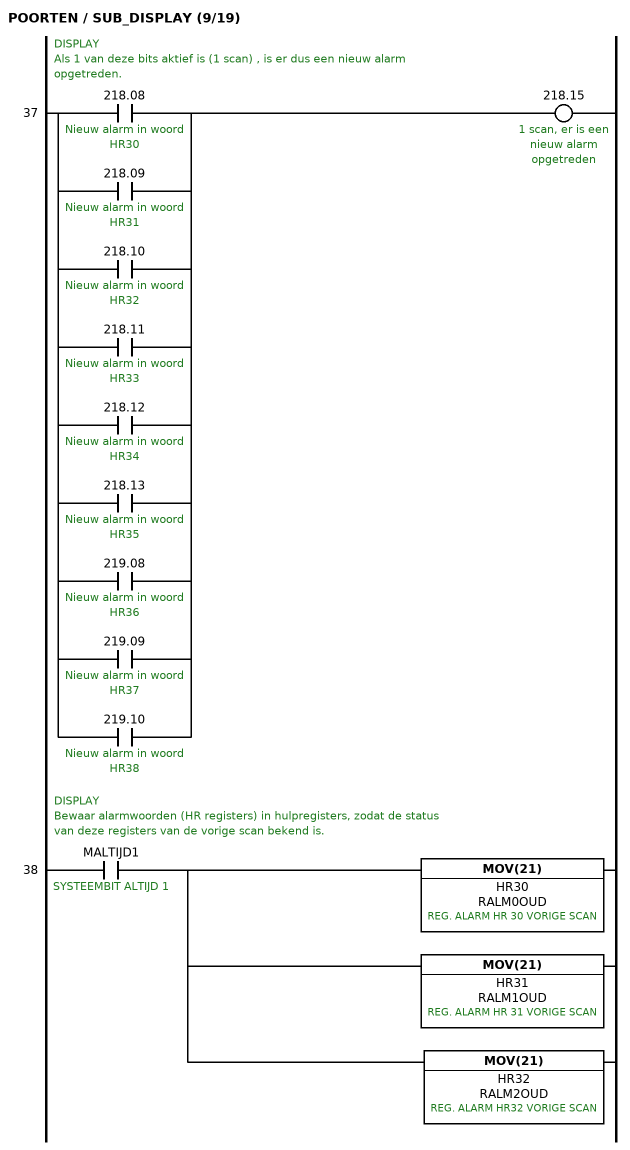
; rung 37: DISPLAY / Als 1 van deze bits aktief is (1 scan) , is er dus een nieuw alarm / opgetreden.
LD 218.08  ; Nieuw alarm in woord HR30
OR 218.09  ; Nieuw alarm in woord HR31
OR 218.10  ; Nieuw alarm in woord HR32
OR 218.11  ; Nieuw alarm in woord HR33
OR 218.12  ; Nieuw alarm in woord HR34
OR 218.13  ; Nieuw alarm in woord HR35
OR 219.08  ; Nieuw alarm in woord HR36
OR 219.09  ; Nieuw alarm in woord HR37
OR 219.10  ; Nieuw alarm in woord HR38
OUT 218.15  ; 1 scan, er is een nieuw alarm opgetreden
; rung 38: DISPLAY / Bewaar alarmwoorden (HR registers) in hulpregisters, zodat de status / van deze registers van de vorige scan bekend is.
LD MALTIJD1  ; SYSTEEMBIT ALTIJD 1
MOV(21) HR30 RALM0OUD  ; REG. ALARM HR 30 VORIGE SCAN
MOV(21) HR31 RALM1OUD  ; REG. ALARM HR 31 VORIGE SCAN
MOV(21) HR32 RALM2OUD  ; REG. ALARM HR32 VORIGE SCAN

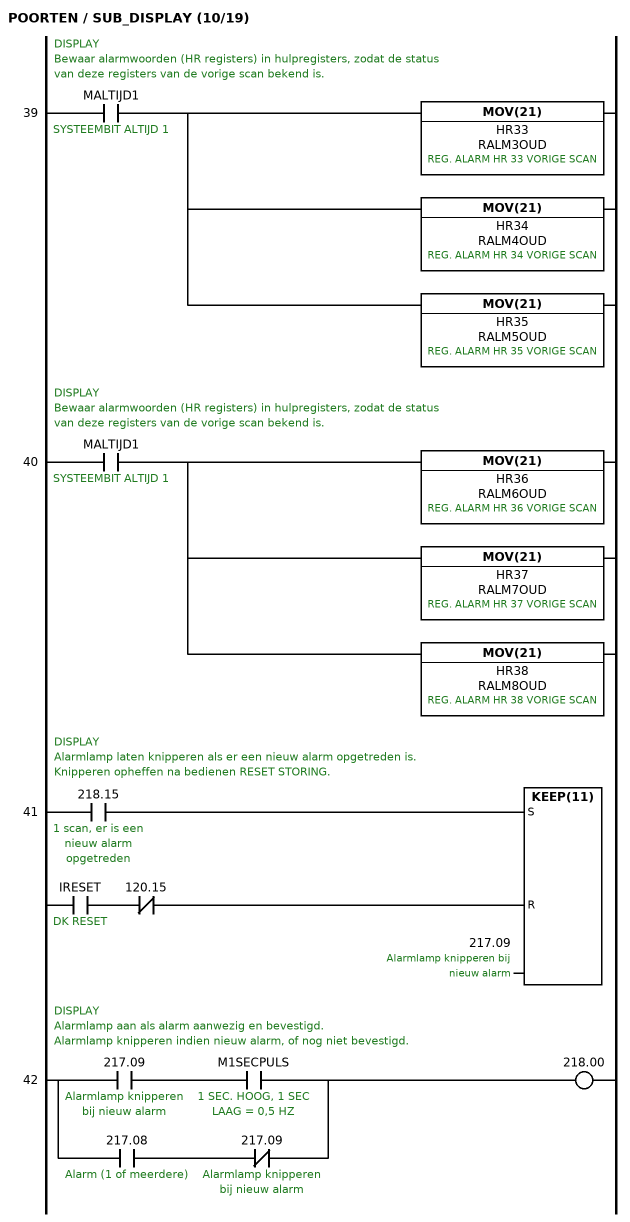
; rung 39: DISPLAY / Bewaar alarmwoorden (HR registers) in hulpregisters, zodat de status / van deze registers van de vorige scan bekend is.
LD MALTIJD1  ; SYSTEEMBIT ALTIJD 1
MOV(21) HR33 RALM3OUD  ; REG. ALARM HR 33 VORIGE SCAN
MOV(21) HR34 RALM4OUD  ; REG. ALARM HR 34 VORIGE SCAN
MOV(21) HR35 RALM5OUD  ; REG. ALARM HR 35 VORIGE SCAN
; rung 40: DISPLAY / Bewaar alarmwoorden (HR registers) in hulpregisters, zodat de status / van deze registers van de vorige scan bekend is.
LD MALTIJD1  ; SYSTEEMBIT ALTIJD 1
MOV(21) HR36 RALM6OUD  ; REG. ALARM HR 36 VORIGE SCAN
MOV(21) HR37 RALM7OUD  ; REG. ALARM HR 37 VORIGE SCAN
MOV(21) HR38 RALM8OUD  ; REG. ALARM HR 38 VORIGE SCAN
; rung 41: DISPLAY / Alarmlamp laten knipperen als er een nieuw alarm opgetreden is. / Knipperen opheffen na bedienen RESET STORING.
LD 218.15  ; 1 scan, er is een nieuw alarm opgetreden
LD IRESET  ; DK RESET
ANDNOT 120.15
KEEP(11) 217.09  ; Alarmlamp knipperen bij nieuw alarm
; rung 42: DISPLAY / Alarmlamp aan als alarm aanwezig en bevestigd. / Alarmlamp knipperen indien nieuw alarm, of nog niet bevestigd.
LD 217.09  ; Alarmlamp knipperen bij nieuw alarm
AND M1SECPULS  ; 1 SEC. HOOG, 1 SEC LAAG = 0,5 HZ
LD 217.08  ; Alarm (1 of meerdere)
ANDNOT 217.09  ; Alarmlamp knipperen bij nieuw alarm
ORLD
OUT 218.00

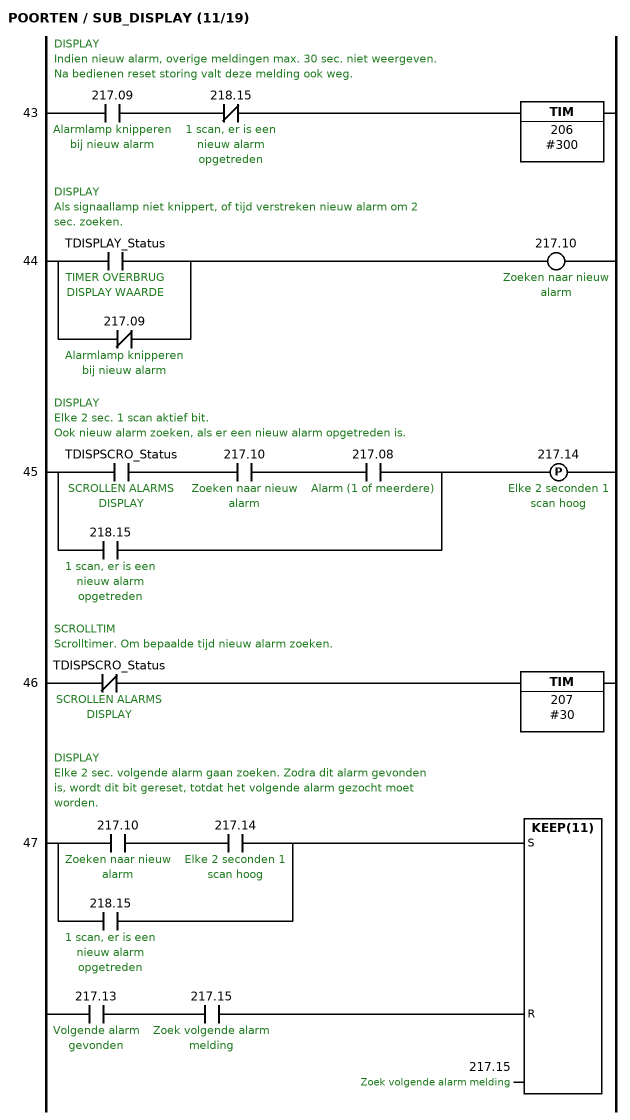
; rung 43: DISPLAY / Indien nieuw alarm, overige meldingen max. 30 sec. niet weergeven. / Na bedienen reset storing valt deze melding ook weg.
LD 217.09  ; Alarmlamp knipperen bij nieuw alarm
ANDNOT 218.15  ; 1 scan, er is een nieuw alarm opgetreden
TIM 206 #300
; rung 44: DISPLAY / Als signaallamp niet knippert, of tijd verstreken nieuw alarm om 2 / sec. zoeken.
LD TDISPLAY_Status  ; TIMER OVERBRUG DISPLAY WAARDE
ORNOT 217.09  ; Alarmlamp knipperen bij nieuw alarm
OUT 217.10  ; Zoeken naar nieuw alarm
; rung 45: DISPLAY / Elke 2 sec. 1 scan aktief bit. / Ook nieuw alarm zoeken, als er een nieuw alarm opgetreden is.
LD TDISPSCRO_Status  ; SCROLLEN ALARMS DISPLAY
AND 217.10  ; Zoeken naar nieuw alarm
AND 217.08  ; Alarm (1 of meerdere)
OR 218.15  ; 1 scan, er is een nieuw alarm opgetreden
DIFU(13) 217.14  ; Elke 2 seconden 1 scan hoog
; rung 46: SCROLLTIM / Scrolltimer. Om bepaalde tijd nieuw alarm zoeken.
LDNOT TDISPSCRO_Status  ; SCROLLEN ALARMS DISPLAY
TIM 207 #30
; rung 47: DISPLAY / Elke 2 sec. volgende alarm gaan zoeken. Zodra dit alarm gevonden / is, wordt dit bit gereset, totdat het volgende alarm gezocht moet / worden.
LD 217.10  ; Zoeken naar nieuw alarm
AND 217.14  ; Elke 2 seconden 1 scan hoog
OR 218.15  ; 1 scan, er is een nieuw alarm opgetreden
LD 217.13  ; Volgende alarm gevonden
AND 217.15  ; Zoek volgende alarm melding
KEEP(11) 217.15  ; Zoek volgende alarm melding

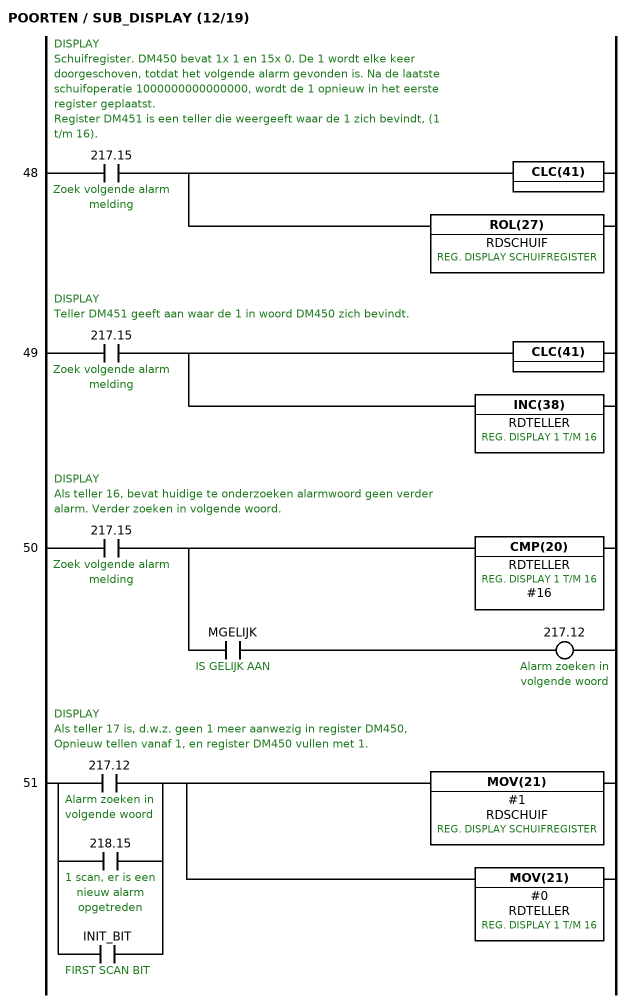
; rung 48: DISPLAY / Schuifregister. DM450 bevat 1x 1 en 15x 0. De 1 wordt elke keer / doorgeschoven, totdat het volgende alarm gevonden is. Na de laatste / schuifoperatie 1000000000000000, wordt de 1 opnieuw in het eerste / register geplaatst. / Register DM451 is een teller die weergeeft waar de 1 zich bevindt, (1 / t/m 16).
LD 217.15  ; Zoek volgende alarm melding
CLC(41)
ROL(27) RDSCHUIF  ; REG. DISPLAY SCHUIFREGISTER
; rung 49: DISPLAY / Teller DM451 geeft aan waar de 1 in woord DM450 zich bevindt.
LD 217.15  ; Zoek volgende alarm melding
CLC(41)
INC(38) RDTELLER  ; REG. DISPLAY 1 T/M 16
; rung 50: DISPLAY / Als teller 16, bevat huidige te onderzoeken alarmwoord geen verder / alarm. Verder zoeken in volgende woord.
LD 217.15  ; Zoek volgende alarm melding
CMP(20) RDTELLER #16  ; REG. DISPLAY 1 T/M 16
AND MGELIJK  ; IS GELIJK AAN
OUT 217.12  ; Alarm zoeken in volgende woord
; rung 51: DISPLAY / Als teller 17 is, d.w.z. geen 1 meer aanwezig in register DM450, / Opnieuw tellen vanaf 1, en register DM450 vullen met 1.
LD 217.12  ; Alarm zoeken in volgende woord
OR 218.15  ; 1 scan, er is een nieuw alarm opgetreden
OR INIT_BIT  ; FIRST SCAN BIT
MOV(21) #1 RDSCHUIF  ; REG. DISPLAY SCHUIFREGISTER
MOV(21) #0 RDTELLER  ; REG. DISPLAY 1 T/M 16

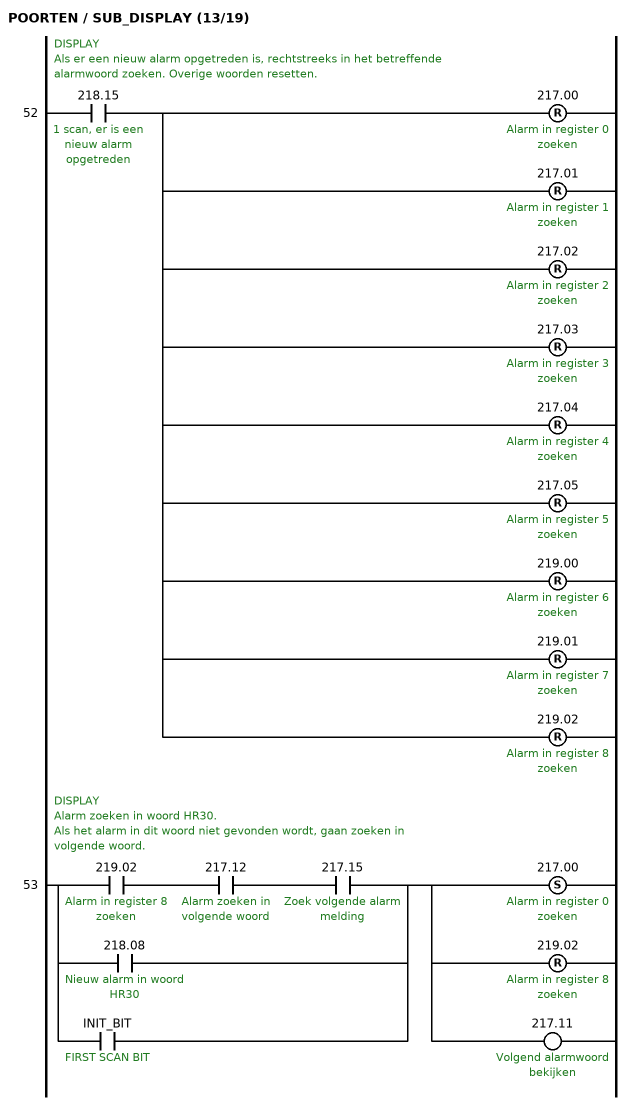
; rung 52: DISPLAY / Als er een nieuw alarm opgetreden is, rechtstreeks in het betreffende / alarmwoord zoeken. Overige woorden resetten.
LD 218.15  ; 1 scan, er is een nieuw alarm opgetreden
RSET 217.00  ; Alarm in register 0 zoeken
RSET 217.01  ; Alarm in register 1 zoeken
RSET 217.02  ; Alarm in register 2 zoeken
RSET 217.03  ; Alarm in register 3 zoeken
RSET 217.04  ; Alarm in register 4 zoeken
RSET 217.05  ; Alarm in register 5 zoeken
RSET 219.00  ; Alarm in register 6 zoeken
RSET 219.01  ; Alarm in register 7 zoeken
RSET 219.02  ; Alarm in register 8 zoeken
; rung 53: DISPLAY / Alarm zoeken in woord HR30. / Als het alarm in dit woord niet gevonden wordt, gaan zoeken in / volgende woord.
LD 219.02  ; Alarm in register 8 zoeken
AND 217.12  ; Alarm zoeken in volgende woord
AND 217.15  ; Zoek volgende alarm melding
OR 218.08  ; Nieuw alarm in woord HR30
OR INIT_BIT  ; FIRST SCAN BIT
SET 217.00  ; Alarm in register 0 zoeken
RSET 219.02  ; Alarm in register 8 zoeken
OUT 217.11  ; Volgend alarmwoord bekijken

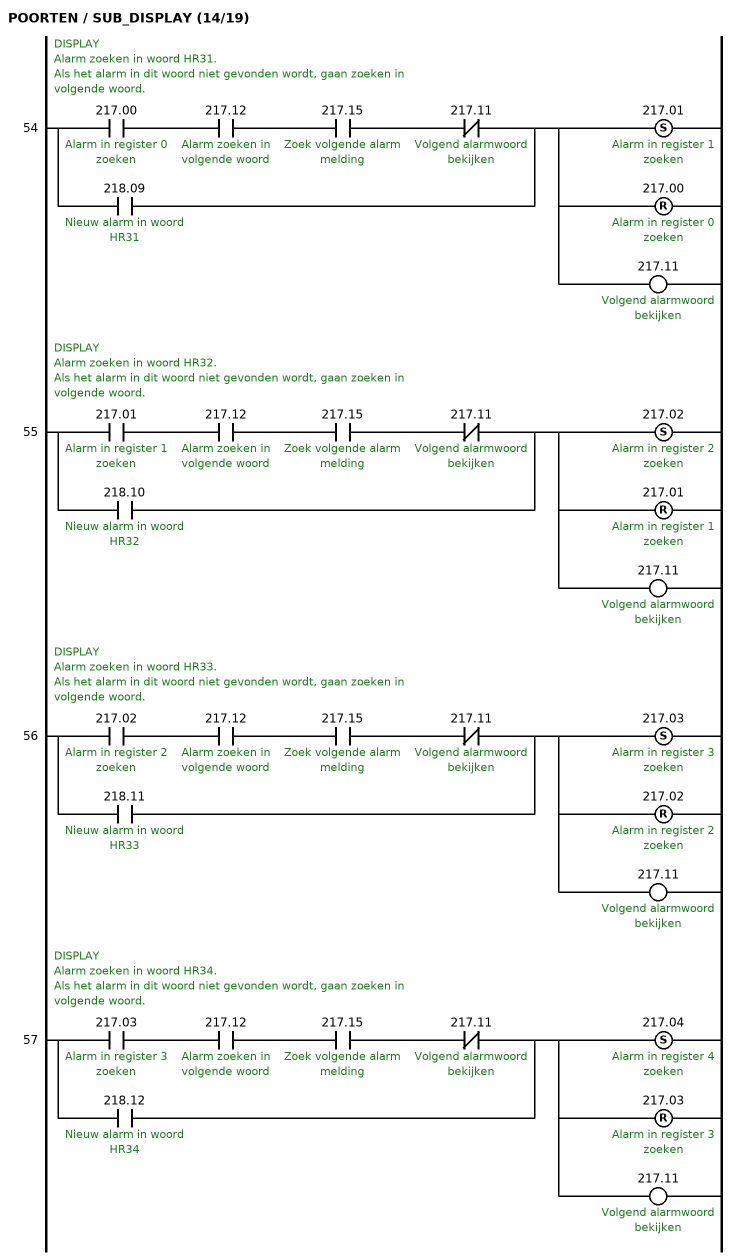
; rung 54: DISPLAY / Alarm zoeken in woord HR31. / Als het alarm in dit woord niet gevonden wordt, gaan zoeken in / volgende woord.
LD 217.00  ; Alarm in register 0 zoeken
AND 217.12  ; Alarm zoeken in volgende woord
AND 217.15  ; Zoek volgende alarm melding
ANDNOT 217.11  ; Volgend alarmwoord bekijken
OR 218.09  ; Nieuw alarm in woord HR31
SET 217.01  ; Alarm in register 1 zoeken
RSET 217.00  ; Alarm in register 0 zoeken
OUT 217.11  ; Volgend alarmwoord bekijken
; rung 55: DISPLAY / Alarm zoeken in woord HR32. / Als het alarm in dit woord niet gevonden wordt, gaan zoeken in / volgende woord.
LD 217.01  ; Alarm in register 1 zoeken
AND 217.12  ; Alarm zoeken in volgende woord
AND 217.15  ; Zoek volgende alarm melding
ANDNOT 217.11  ; Volgend alarmwoord bekijken
OR 218.10  ; Nieuw alarm in woord HR32
SET 217.02  ; Alarm in register 2 zoeken
RSET 217.01  ; Alarm in register 1 zoeken
OUT 217.11  ; Volgend alarmwoord bekijken
; rung 56: DISPLAY / Alarm zoeken in woord HR33. / Als het alarm in dit woord niet gevonden wordt, gaan zoeken in / volgende woord.
LD 217.02  ; Alarm in register 2 zoeken
AND 217.12  ; Alarm zoeken in volgende woord
AND 217.15  ; Zoek volgende alarm melding
ANDNOT 217.11  ; Volgend alarmwoord bekijken
OR 218.11  ; Nieuw alarm in woord HR33
SET 217.03  ; Alarm in register 3 zoeken
RSET 217.02  ; Alarm in register 2 zoeken
OUT 217.11  ; Volgend alarmwoord bekijken
; rung 57: DISPLAY / Alarm zoeken in woord HR34. / Als het alarm in dit woord niet gevonden wordt, gaan zoeken in / volgende woord.
LD 217.03  ; Alarm in register 3 zoeken
AND 217.12  ; Alarm zoeken in volgende woord
AND 217.15  ; Zoek volgende alarm melding
ANDNOT 217.11  ; Volgend alarmwoord bekijken
OR 218.12  ; Nieuw alarm in woord HR34
SET 217.04  ; Alarm in register 4 zoeken
RSET 217.03  ; Alarm in register 3 zoeken
OUT 217.11  ; Volgend alarmwoord bekijken

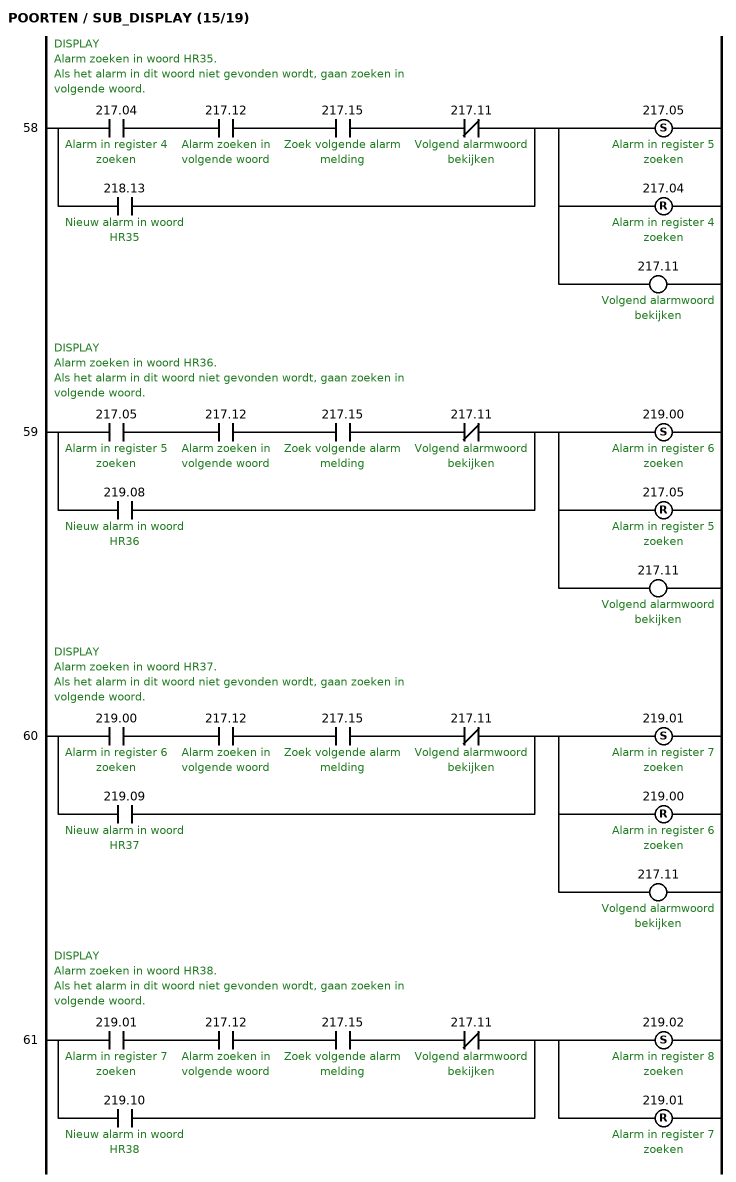
; rung 58: DISPLAY / Alarm zoeken in woord HR35. / Als het alarm in dit woord niet gevonden wordt, gaan zoeken in / volgende woord.
LD 217.04  ; Alarm in register 4 zoeken
AND 217.12  ; Alarm zoeken in volgende woord
AND 217.15  ; Zoek volgende alarm melding
ANDNOT 217.11  ; Volgend alarmwoord bekijken
OR 218.13  ; Nieuw alarm in woord HR35
SET 217.05  ; Alarm in register 5 zoeken
RSET 217.04  ; Alarm in register 4 zoeken
OUT 217.11  ; Volgend alarmwoord bekijken
; rung 59: DISPLAY / Alarm zoeken in woord HR36. / Als het alarm in dit woord niet gevonden wordt, gaan zoeken in / volgende woord.
LD 217.05  ; Alarm in register 5 zoeken
AND 217.12  ; Alarm zoeken in volgende woord
AND 217.15  ; Zoek volgende alarm melding
ANDNOT 217.11  ; Volgend alarmwoord bekijken
OR 219.08  ; Nieuw alarm in woord HR36
SET 219.00  ; Alarm in register 6 zoeken
RSET 217.05  ; Alarm in register 5 zoeken
OUT 217.11  ; Volgend alarmwoord bekijken
; rung 60: DISPLAY / Alarm zoeken in woord HR37. / Als het alarm in dit woord niet gevonden wordt, gaan zoeken in / volgende woord.
LD 219.00  ; Alarm in register 6 zoeken
AND 217.12  ; Alarm zoeken in volgende woord
AND 217.15  ; Zoek volgende alarm melding
ANDNOT 217.11  ; Volgend alarmwoord bekijken
OR 219.09  ; Nieuw alarm in woord HR37
SET 219.01  ; Alarm in register 7 zoeken
RSET 219.00  ; Alarm in register 6 zoeken
OUT 217.11  ; Volgend alarmwoord bekijken
; rung 61: DISPLAY / Alarm zoeken in woord HR38. / Als het alarm in dit woord niet gevonden wordt, gaan zoeken in / volgende woord.
LD 219.01  ; Alarm in register 7 zoeken
AND 217.12  ; Alarm zoeken in volgende woord
AND 217.15  ; Zoek volgende alarm melding
ANDNOT 217.11  ; Volgend alarmwoord bekijken
OR 219.10  ; Nieuw alarm in woord HR38
SET 219.02  ; Alarm in register 8 zoeken
RSET 219.01  ; Alarm in register 7 zoeken

